// TwinCAT 3 PLC project PMPS_Prototype_Arbiter
// ProgramVersion: 3.1.4022.1
// libraries:
//   LCLS General, * (SLAC)
//   Tc2_MC2, * (Beckhoff Automation GmbH)
//   Tc2_Standard, * (Beckhoff Automation GmbH)
//   Tc2_System, * (Beckhoff Automation GmbH)
//   Tc2_Utilities, * (Beckhoff Automation GmbH)
//   Tc3_Module, * (Beckhoff Automation GmbH)
//   VisuDialogs, * (System)
//   VisuSymbols,3.5.10.0,System
// project tree:
//   DUTs/ E_ExampleDeviceStates.TcDUT (not stored), ST_BeamParams.TcDUT, ST_BinarySolidAttenuator.TcDUT (not stored), ST_Device.TcDUT, ST_DeviceState.TcDUT, ST_SolidAttenuatorBlade.TcDUT
//   / GlobalTextList.TcGTLO, ImagePool.TcIPO (not stored), PlcTask.TcTTO (not stored), Visualization Manager.TcVMO (not stored)
//   GVLs/ GVL.TcGVL, PMPS_GVL_BeamParams.TcGVL
//   POUs/DeviceImplementationEx1/ FB_ExampleDevice.TcPOU (not stored), FB_ExampleDeviceSM.TcPOU (not stored)
//   POUs/DeviceImplementationEx2/ FB_ExampleDeviceSM_All.TcPOU
//   POUs/HelperFunctions/ F_DifferentBeamParams.TcPOU (not stored), F_SafeBPCompare.TcPOU (not stored), F_SetBeamParams.TcPOU (not stored), F_SetStateParams.TcPOU (not stored)
//   POUs/ MAIN.TcPOU, PMPS_Arbiter.TcPOU
//   POUs/MajorComponents/ FB_BeamClassOutputs.TcPOU, FB_LinearGovernor.TcPOU, BeamParameterTransitionManager.TcPOU (not stored), FB_Arbiter.TcPOU, FB_BeamParamAssertionPool.TcPOU (not stored), FB_LinearDeviceStateTable.TcPOU (not stored)
//   POUs/TestComponents/ FB_AttenuatorSimulator.TcPOU, FB_MachineSimulator.TcPOU (not stored), FB_SolidAttenuator.TcPOU
//   VISUs/ ImagerGUI.TcVIS, Visualization.TcVIS
// real-time tasks:
//   TASK PlcTask: cycle T#1ms, priority 20, ADS port 350
// motion (NC):
//   TASK NC-Task 1 SAF: cycle T#2ms, priority 4, ADS port 501
//   TASK NC-Task 1 SVB: cycle T#10ms, priority 8, ADS port 511
//   AXIS Dev1 (id 1)
//   AXIS Dev 2 (id 2)
// variable links:
//   PMPS_Prototype_Arbiter/PMPS_Prototype_Arbiter Instance <-> NC-Task 1 SAF/Axes/Dev 2
//     PlcTask Inputs/MAIN.fbDev2.stDevice.stAxis.NcToPlc <-> Outputs/ToPlc
//     PlcTask Outputs/MAIN.fbDev2.stDevice.stAxis.PlcToNc <-> Inputs/FromPlc
//   PMPS_Prototype_Arbiter/PMPS_Prototype_Arbiter Instance <-> NC-Task 1 SAF/Axes/Dev1
//     PlcTask Inputs/MAIN.fbDev1.stDevice.stAxis.NcToPlc <-> Outputs/ToPlc
//     PlcTask Outputs/MAIN.fbDev1.stDevice.stAxis.PlcToNc <-> Inputs/FromPlc

// ---- DUTs/ST_BeamParams.TcDUT
TYPE ST_BeamParams :
STRUCT
	// Beam parameters
	// These must be filled in by the caller.
	
	//Note: fAtt is a local parameter, meaning it is distributed to the nearest
	// upstream attenuator component.
	fAtt : REAL := 100; //Requested attenuation %
	
	
	
	//Machine parameters
	nBeamClass	:	BYTE := 16#F;
	nRate	:	UDINT	:= 10; //Pulse-rate
	fPP_mJ : REAL := 20; //Per pulse max energy (mJ)
	fUpper_eV	:	REAL	:= 20000; //Requested max eV
	fLower_eV	:	REAL	:= 0; //Requested lower eV
	reV	:	REAL	:=0; //Photon energy (calculated by undulator gap)
END_STRUCT
END_TYPE

// ---- DUTs/ST_Device.TcDUT
TYPE ST_Device :
STRUCT
	//IO
	stAxis	:	AXIS_REF;
	//The following limit switches must be TRUE or high (ie. NC) to enable that direction of motion
	//The EPICS display should show an inverted indicator to communicate end of travel reached
	i_xLoLim	AT %I*	:	BOOL; //Wire normally-closed
	i_xHiLim	AT %I*	:	BOOL; //Wire normally-closed
	
	//Acuator Parameters
	lrUpperPositionLimit	:	LREAL := 10000000000; //Use in conjuntion with limit switches or set to a huge number to ignore
	lrLowerPositionLimit	:	LREAL := -10000000000; //Use in conjuntion with limit switches or set to a huge number to ignore
	
	xEnable	:	BOOL := TRUE;
	
	//Supervisory System
	
	//MPS Override
	xOverrideMPSLimits	: BOOL := FALSE; //Set true to move beyond MPS limits. Note this will trip beam off.
	
	//Device States
	StateTable		:	FB_LinearDeviceStateTable;
	//astStates	:	ARRAY[0..PMPS_GVL_BeamParams.cnMaxStateArrayLen] OF	ST_DeviceState;
	
	stTransitionState	:	ST_DeviceState; //The transition state might have non-zero beam parameters
	nSafeState			:	UDINT; //State where the device is considered safe
	nTransitionState	:	UDINT;
	
	nRequestedState	:	UDINT; //EPICS control, cleaned (checked against array limits) and deposited in nTargetState
	nTargetState	:	UDINT; //The requested state should be deposited here after cleaning
	nActiveState	:	UDINT; //The last successfully reached state
	
	
END_STRUCT
END_TYPE

// ---- DUTs/ST_DeviceState.TcDUT
TYPE ST_DeviceState :
STRUCT
	
	//Database key
	
	//Parent Device
	sParentDevice	:	STRING;
	
	//State name
	sStateName	:	STRING;
	nStateRef	:	UDINT; //Primary key of device state database
	
	//////////////////
	// This stuff may belong in a sub-class or something
	//Position
	rPosition	:	REAL := 0;
	//Tolerance
	rTolerance :	REAL := 0; //+/- amount
	//////////////////
	//Required beam parameters
	stReqBeamParam	:	ST_BeamParams;

END_STRUCT
END_TYPE

// ---- DUTs/ST_SolidAttenuatorBlade.TcDUT
TYPE ST_SolidAttenuatorBlade :
STRUCT
	xRequestedIn	:	BOOL;
	xCurrentIn	:	BOOL;
	rThickness	:	REAL;
END_STRUCT
END_TYPE

// ---- GVLs/GVL.TcGVL

VAR_GLOBAL
	fbArbiter	:	FB_Arbiter;
	g_rTestingVelocity	:	LREAL := VISIBLE_TEST_VELOCITY;
END_VAR

VAR_GLOBAL CONSTANT
	EXCLUDED_ASSERTION_ID	:	UDINT	:= 16#FFFFFFFF; //An assertion ID that should always return "not found" in the assertion pool
	VISIBLE_TEST_VELOCITY	:	LREAL	:= 10;
	FAST_TEST_VELOCITY		:	LREAL	:= 100;
	MAX_DEVICE_STATES		:	UDINT	:= 300;
END_VAR

// ---- GVLs/PMPS_GVL_BeamParams.TcGVL
{attribute 'qualified_only'}
VAR_GLOBAL
	stReqFBDBeamParamsSum	:	ST_BeamParams;
	stReqMethBeamParamSum	:	ST_BeamParams;
	stCurrentBeamParameters	:	ST_BeamParams;
END_VAR
VAR_GLOBAL CONSTANT
	cstFullBeam	:	ST_BeamParams := (
		fAtt := 0,
		fPP_mJ := 1E4,
		fUpper_eV := 1E4,
		fLower_eV := 0,
		nRate	:= UDINT#1000000,
		
);
	cstSafeBeam	:	ST_BeamParams := (
		fAtt := 100,
		fPP_mJ := 0,
		fUpper_eV := 0,
		fLower_eV := 0,
		nRate	:= 0
);
	cnMaxStateArrayLen : INT := 20;
	
	MAX_ASSERIONS	:	UDINT := 100; //Maximum number of assertions permitted in the arbiter
END_VAR

// ---- POUs/MajorComponents/FB_Arbiter.TcPOU
(* FB Arbiter

The arbiter primary objectives are:
- Provide a simple interface for devices to request beam parameter sets
- Provide a way for devices to verify their BPS is active in the arbiter
- Provide a way for devices remove their requests from evaluation
- Evaluate all active beam parameter requests registered with the aribiter,
to determine the safest combination of all sets, provide this set as an output.
- Do all of this with minimal overhead

To these ends, the arbiter uses a hash-table, the rows being a state-id as the key, and a corresponding
 beam parameter set to be evaluated against all the other sets (or rows), in the table.
 
The hash table can be thought of as an array on steriods, they are worth reading about, suffice to say
the hash table will tell you when you reach the end of all the entries, and enables us to find entries quickly.

These features efficiently address the addition, removal, and verification of beam parameter sets listed in the above requirements.

An important thing to pay attention to is the A_Arbitrate action. This action implements the evaluation of beam parameter
sets against each other.

*)

FUNCTION_BLOCK FB_Arbiter
VAR_INPUT
	i_nStateID	:	UDINT; //Set to the stateID of the state requesting the beam parameter set
	i_stAssertBeamParams	:	ST_BeamParams; //Set to the beam parameter set of the state required
END_VAR
VAR_OUTPUT
	q_stBeamParams	:	ST_BeamParams; //Updated on each cycle of the arbiter FB with the current arbitrated beam parameter set
	
	q_xStateIDFound	:	BOOL; //Set true if a state-id is found in the assertion pool after calling A_VerifyAssertion
END_VAR
VAR
	
	fbBPAssertionPool	:	FB_BeamParamAssertionPool; //Table of active beam parameter assertions
	
	getPosPtr	: POINTER TO T_HashTableEntry := 0; 
	getBPStruct	:	ST_BeamParams;
	stOutputBP	:	ST_BeamParams; //Safest beam parameters from all in the assertion pool
	
	
END_VAR

//Arbitrate
(*
This step cycles through every hash table entry, comparing
the beam parameters from each assertion to what we're planning
to assert.

The safer of the two parameters is kept so at the end we may
have a mix of beam parameters, the composition being safe for
all asserters.

*)

//Safest parameters to start
stOutputBP := F_SetBeamParams(
	fAtt := 100,
	fPP_mJ := 0,
	fLower_eV := 0,
	fUpper_eV := 1800,
	nRate := 0
	);

fbBPAssertionPool.A_GetFirst( putPosPtr := 0, getPosPtr=>getPosPtr, getValue=>getBPStruct );
IF fbBPAssertionPool.bOk THEN
	
	//The first entry in the hash table is taken as the setting to arbitrate against
	stOutputBP := F_SetBeamParams(
		fAtt := getBPStruct.fAtt,
		fPP_mJ := getBPStruct.fPP_mJ,
		fLower_eV := getBPStruct.fLower_eV,
		fUpper_eV := getBPStruct.fUpper_eV,
		nRate := getBPStruct.nRate
	);

	REPEAT
		fbBPAssertionPool.A_GetNext( putPosPtr := fbBPAssertionPool.getPosPtr , getPosPtr=>getPosPtr, getValue=>getBPStruct );
		IF fbBPAssertionPool.bOk THEN
			A_Arbitrate();
		END_IF
	UNTIL NOT fbBPAssertionPool.bOk
	END_REPEAT

END_IF

q_stBeamParams := stOutputBP;

ACTION A_Arbitrate:

//Attenuation
//Add something here to register the key that won for each param
stOutputBP.fAtt := MAX(stOutputBP.fAtt, getBPStruct.fAtt);

//Pulse energy
stOutputBP.fPP_mJ := MIN(stOutputBP.fPP_mJ, getBPStruct.fPP_mJ);

//Photon energy ranges
stOutputBP.neVReqRange := stOutputBP.neVReqRange AND getBPStruct.neVReqRange;

//Rate
stOutputBP.nRate := MIN(stOutputBP.nRate, getBPStruct.nRate);
END_ACTION

ACTION A_AssertBP:
//fbTable.A_Add( key := 12345, putValue := putValue, getPosPtr=>getPosPtr, getValue=>getValue );

(* This action adds a state-id and beam parameter set to the beam parameter assertion pool (arbiter
hash table). Use like so:

fbArbiter.A_AssertBP(
i_nStateID := nStateID,
i_stAssertBeamParams := stDesiredBeamParams
);

*)

IF i_nStateID <> EXCLUDED_ASSERTION_ID THEN

	fbBPAssertionPool.A_Add(
		key := i_nStateID,
		putValue := i_stAssertBeamParams,
		getPosPtr=>getPosPtr,
		getValue => getBPStruct
	);
END_IF
	
IF NOT fbBPAssertionPool.bOk THEN
	; //Overflow <TODO>
END_IF
END_ACTION

ACTION A_Init:
// Clears the entire beam parameter assertion pool (hashtable).

fbBPAssertionPool.A_Reset();
END_ACTION

ACTION A_RemoveAssertion:

(* Searches for a state-id, and removes it from the assertion pool.

Use like so:
fbArbiter.A_RemoveAssertion(
i_nStateId := nStateIDAssertionToRemove
);

*)

IF i_nStateId <> EXCLUDED_ASSERTION_ID THEN
	fbBPAssertionPool.A_Remove(key := i_nStateId, getPosPtr=>getPosPtr, getValue=>getBPStruct);
	
	IF fbBPAssertionPool.bOk THEN
		;
	ELSE
		;
	END_IF
END_IF
END_ACTION

ACTION A_VerifyAssertion:

(* Searches state assertion pool for a state-id, and sets q_xStateIDFound true if found.

Use like so:

fbArbiter.A_VerifyAssertion(
i_nStateId := nStateIDAssertionToCheck
);

IF fbArbiter.q_xStateIDFound THEN:
	Do something
ELSE:
	Don't do something

*)

IF i_nStateID <> EXCLUDED_ASSERTION_ID THEN
	
	fbBPAssertionPool.A_Lookup( key := i_nStateID, getPosPtr=>getPosPtr, getValue=>getBPStruct );

	q_xStateIDFound	:= fbBPAssertionPool.bOk;

ELSE
	q_xStateIDFound := FALSE;
END_IF
END_ACTION

END_FUNCTION_BLOCK

// ---- POUs/DeviceImplementationEx2/FB_ExampleDeviceSM_All.TcPOU
(* This version of the block is self contained. Minimizes wiring.*)
FUNCTION_BLOCK FB_ExampleDeviceSM_All
VAR_INPUT
	cBase: UDINT;
END_VAR
VAR_OUTPUT
END_VAR
VAR_IN_OUT
	
END_VAR
VAR
	stDevice	:	ST_Device;
	fbGovernor	:	FB_LinearGovernor;
	mcPower	:	MC_Power;
	mcStop: MC_Stop;
	mcAbsolute	:	MC_MoveAbsolute;
	fbBPTM	:	BeamParameterTransitionManager;
	xStartMove: BOOL;
	
	stCheckState: ST_DeviceState;
	stTargetState	:	ST_DeviceState; //Target device state

END_VAR
VAR PERSISTENT
	nLastActiveState	:	UDINT;
END_VAR

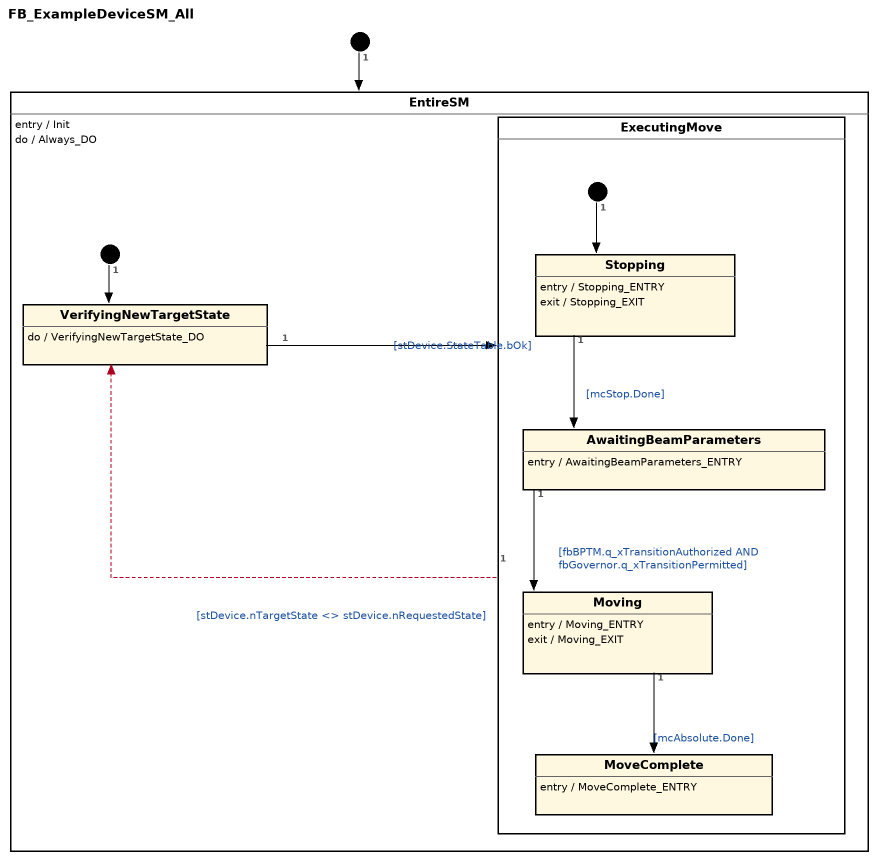
STATECHART FB_ExampleDeviceSM_All  // abortable
    START StartState3
    COMPOSITE STATE EntireSM
        entry / Init
        do / Always_DO
        START StartState1
        COMPOSITE STATE ExecutingMove
            START StartState2
            STATE Stopping
                entry / Stopping_ENTRY
                exit / Stopping_EXIT
            STATE AwaitingBeamParameters
                entry / AwaitingBeamParameters_ENTRY
            STATE Moving
                entry / Moving_ENTRY
                exit / Moving_EXIT
            STATE MoveComplete
                entry / MoveComplete_ENTRY
            StartState2 -> Stopping  // priority 1, on completion
            Stopping -> AwaitingBeamParameters [mcStop.Done] // priority 1, rising edge
            AwaitingBeamParameters -> Moving [fbBPTM.q_xTransitionAuthorized AND fbGovernor.q_xTransitionPermitted] // priority 1, rising edge
            Moving -> MoveComplete [mcAbsolute.Done] // priority 1, rising edge
        END_STATE
        STATE VerifyingNewTargetState
            do / VerifyingNewTargetState_DO
        StartState1 -> VerifyingNewTargetState  // priority 1, on completion
        ExecutingMove -> VerifyingNewTargetState [stDevice.nTargetState <> stDevice.nRequestedState] // priority 1, exception, rising edge
        VerifyingNewTargetState -> ExecutingMove [stDevice.StateTable.bOk] // priority 1
    END_STATE
    StartState3 -> EntireSM  // priority 1, on completion
END_STATECHART

ACTION Always_DO:
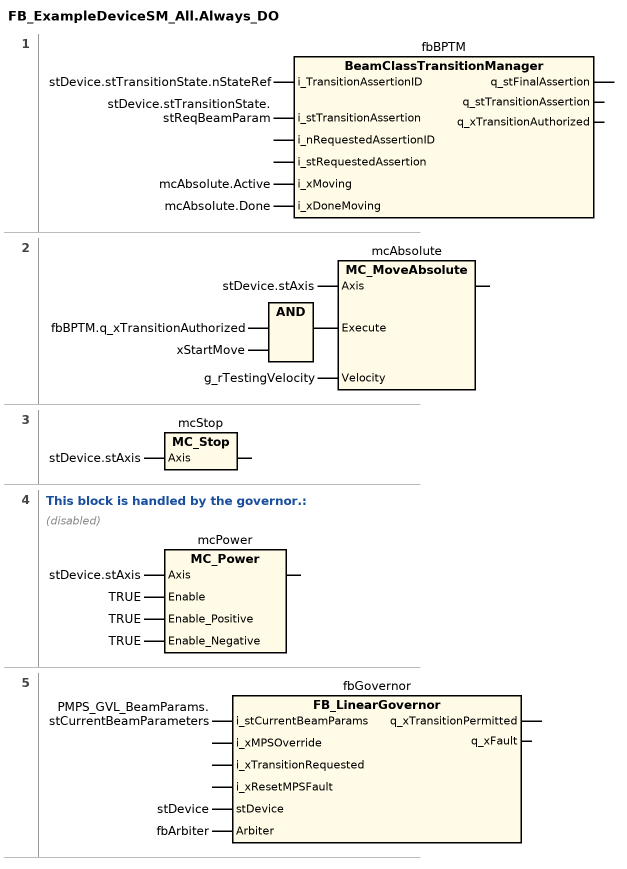
// NETWORK 1
fbBPTM(
    i_TransitionAssertionID := stDevice.stTransitionState.nStateRef,
    i_stTransitionAssertion := stDevice.stTransitionState.stReqBeamParam,
    i_xMoving := mcAbsolute.Active,
    i_xDoneMoving := mcAbsolute.Done); // BeamClassTransitionManager

// NETWORK 2
mcAbsolute(
    Axis := stDevice.stAxis,
    Execute := fbBPTM.q_xTransitionAuthorized AND xStartMove,
    Velocity := g_rTestingVelocity); // MC_MoveAbsolute

// NETWORK 3
mcStop(Axis := stDevice.stAxis); // MC_Stop

// NETWORK 4 (disabled)
// label: This block is handled by the governor.
// mcPower(Axis := stDevice.stAxis, Enable := TRUE, Enable_Positive := TRUE, Enable_Negative := TRUE); // MC_Power

// NETWORK 5
fbGovernor(
    i_stCurrentBeamParams := PMPS_GVL_BeamParams.stCurrentBeamParameters,
    stDevice := stDevice,
    Arbiter := fbArbiter); // FB_LinearGovernor
END_ACTION

ACTION AwaitingBeamParameters_ENTRY:
fbBPTM.i_stRequestedAssertion := stTargetState.stReqBeamParam;
fbBPTM.i_nRequestedAssertionID := stTargetState.nStateRef;

//Tell the governor that we're trying to move.
fbGovernor.i_xTransitionRequested := TRUE;
END_ACTION

ACTION Init:

//Safe State
stDevice.nSafeState := cBase;
stDevice.nTransitionState := cBase+100;

//Initialize the State Table
stDevice.StateTable.A_Reset();

//Device State Table Instantiation
F_SetStateParams(
	nStateRef := stDevice.nSafeState,
	rPosition := 0,
	rTolerance := 10,
	stBeamParams := PMPS_GVL_BeamParams.cstFullBeam,
	Table := stDevice.StateTable
);
F_SetStateParams(
	nStateRef := cBase + 1,
	rPosition := 100,
	rTolerance := 10,
	stBeamParams := F_SetBeamParams(
		fAtt := 20,
		fPP_mJ := 1,
		fLower_eV := 0,
		fUpper_eV := 1500,
		nRate := 10
		),
	Table := stDevice.StateTable
);
F_SetStateParams(
	nStateRef := cBase + 2,
	rPosition := 200,
	rTolerance := 10,
	stBeamParams := F_SetBeamParams(
		fAtt := 30,
		fPP_mJ := 1,
		fLower_eV := 0,
		fUpper_eV := 1500,
		nRate := 10
		),
	Table := stDevice.StateTable
);
F_SetStateParams(
	nStateRef := cBase + 3,
	rPosition := 300,
	rTolerance := 10,
	stBeamParams := F_SetBeamParams(
		fAtt := 20,
		fPP_mJ := 1,
		fLower_eV := 0,
		fUpper_eV := 1500,
		nRate := 10
		),
	Table := stDevice.StateTable
);

F_SetStateParams(
	nStateRef := stDevice.nTransitionState,
	rPosition := 300,
	rTolerance := 10,
	stBeamParams := F_SetBeamParams(
		fAtt := 100,
		fPP_mJ := 0,
		fLower_eV := 0,
		fUpper_eV := 1500,
		nRate := 0
		),
	Table := stDevice.StateTable
);

stDevice.StateTable.A_Lookup(
	key := stDevice.nTransitionState,
	getValue => stDevice.stTransitionState
);

//Need an initialization routine for setting the active state
//Check if the device is at the last known state
//If the device is within the state boundaries, it's considered to be in that state
stDevice.StateTable.A_Lookup(key:= nLastActiveState);
IF stDevice.StateTable.bOk THEN
	stCheckState := stDevice.StateTable.getValue;
ELSE
	stCheckState := stDevice.stTransitionState; //This needs to be safer <TODO>
END_IF

IF stDevice.stAxis.NcToPlc.ActPos <= stCheckstate.rPosition + stCheckState.rTolerance AND
	stDevice.stAxis.NcToPlc.ActPos >= stCheckState.rPosition - stCheckState.rTolerance THEN
	stDevice.nActiveState := nLastActiveState;
ELSE
	stDevice.nActiveState := stDevice.nTransitionState;
END_IF

//Simulation Hardware Limit Switches
stDevice.i_xHiLim := TRUE;
stDevice.i_xLoLim := TRUE;
END_ACTION

ACTION Initialize:

END_ACTION

ACTION MoveComplete_ENTRY:
//Clear transition request
fbGovernor.i_xTransitionRequested := FALSE;
//Latch active state
stDevice.nActiveState := stDevice.nTargetState;
nLastActiveState := stDevice.nActiveState;
END_ACTION

ACTION Moving_ENTRY:
xStartMove := TRUE;
mcAbsolute.Position := stTargetState.rPosition;
END_ACTION

ACTION Moving_EXIT:
xStartMove := FALSE;
END_ACTION

ACTION NewMove_ENTRY:

END_ACTION

ACTION Stopping_ENTRY:
mcStop.Execute := TRUE;
END_ACTION

ACTION Stopping_EXIT:
mcStop.Execute := FALSE;
END_ACTION

ACTION VerifyingNewTargetState_DO:
stDevice.StateTable.A_Lookup(
	key := stDevice.nRequestedState
);

IF stDevice.StateTable.bOk THEN
	stTargetState := stDevice.StateTable.getValue;
	stDevice.nTargetState := stDevice.nRequestedState;
ELSE
	; //log ignored state/ generate an error? <TODO>
END_IF
END_ACTION

END_FUNCTION_BLOCK

// ---- POUs/MajorComponents/FB_LinearGovernor.TcPOU

(* The governor is meant to check your work and keep you from making mistakes.

Checks:
Does your state match the device position and visa versa?
Are the beam parameters safe for the device state?
Did you properly assert the transition and final beam parameters?

*)
FUNCTION_BLOCK FB_LinearGovernor
VAR_INPUT
	i_stCurrentBeamParams	:	ST_BeamParams; //Link to global beam params
	i_xMPSOverride			:	BOOL; //True releases MPS limits after a delay
	i_xTransitionRequested	:	BOOL; //Set true to request a transition
	i_xResetMPSFault	:	BOOL; //Set true to clear MPS fault 
END_VAR
VAR_OUTPUT
	q_xTransitionPermitted	:	BOOL; //True when governor has released restrictions
	q_xFault	:	BOOL; //Set if MC_Power has an error, or override mode is requested
END_VAR
VAR_IN_OUT
	stDevice	:	ST_Device; //The governed
	Arbiter	:	FB_Arbiter;
END_VAR
VAR
	mcPower	:	MC_Power;
	
	xActuatorPositiveEnable: BOOL;
	xActuatorNegativeEnable: BOOL;
	
	xMPSPositiveEnable	:	BOOL;
	xMPSNegativeEnable	:	BOOL;
	lrPosition: LREAL;
	
	lrLatchedTargetPosition	:	LREAL;
	lrLatchedTargetTolerance	:	LREAL;
	
	lrMPSUpperLimit: LREAL;
	lrMPSLowerLimit: LREAL;
	rtNewState: R_TRIG;
	xTransitionOK: BOOL;
	
	tonMPSOverrideMode	:	TON := (
		PT := T#5S
	);
	
	srMPSFault	:	SR;
	// Actuator out of bounds fault
	xActuatorOOB: BOOL;
	//Beam parameters out of spec
	xBeamParamsOOS: BOOL;
	//Beam parameters of currently latched state
	
	stLatchedBeamParams: ST_BeamParams;
	stTargetState: ST_DeviceState;
	
	rtLatchNewState	:	R_TRIG;
	xInit: BOOL := TRUE;
	
	stInitDeviceState: ST_DeviceState;
	// Indicates an error with initialization
	xInitFault: BOOL;
	// Indicates the state could not be found in the state table. There may be something wrong in the device state machine implementation or state table instantiation.
	xStateLookupError: BOOL;
END_VAR


lrPosition := stDevice.stAxis.NcToPlc.ActPos; //Actuator position

stDevice.stAxis.ReadStatus();
//Init
////////////////////////////////
	IF xInit THEN
		xInit := FALSE;
		stDevice.StateTable.A_Lookup(key := stDevice.nActiveState);
		IF stDevice.StateTable.bOk THEN
			stInitDeviceState := stDevice.StateTable.getValue;
			xInitFault := FALSE;
		ELSE
			xInitFault := TRUE;
		END_IF
		lrLatchedTargetPosition := stInitDeviceState.rPosition;
		lrLatchedTargetTolerance := stInitDeviceState.rTolerance;
		stLatchedBeamParams := stInitDeviceState.stReqBeamParam;
	END_IF

// The governor will permit transitions once it verifies the transition assertion is active
// Note the governor does not verify the target state beam params are asserted, perhaps it should <TODO>
////////////////////////////////
	IF i_xTransitionRequested THEN
		Arbiter.A_VerifyAssertion(
			i_nStateID := stDevice.stTransitionState.nStateRef
		);
		xTransitionOK := Arbiter.q_xStateIDFound AND F_SafeBPCompare(PMPS_GVL_BeamParams.stCurrentBeamParameters, stDevice.stTransitionState.stReqBeamParam);
		
		//Set the target state for evaluation in further logic
		stdevice.StateTable.A_Lookup(key := stDevice.nTargetState);
		IF stDevice.StateTable.bOk THEN
			stTargetState := stDevice.StateTable.getValue;
			xStateLookupError := FALSE;
		ELSE
			xStateLookupError := TRUE;
		END_IF
	ELSE
		xTransitionOK := FALSE;
	END_IF

(* Note about TransitionRequested

If TransitionRequested goes false during a transition, an MPS fault may be induced. This occurs
because the Actuator Out of Bounds fault will go back to using the original state limits, which
the axis may have already moved beyond.

To avoid this transient fault, make sure your device state machine is implemented such that the 
transition request to the governor block remains high until the target position is reached.
*)

//Determine if a transition is complete and latch the new state
(* A transition is complete when:

Axis at standstill.
Axis within tolerance.
No transition req.

Once these conditions are met, the MPS limits shall re-engage to restrict the
axis motion to the tolerance around the state position and the MPS fault monitors
shall evaluate based on the newly latched target state.
*)

rtLatchNewState(CLK := stDevice.stAxis.Status.StandStill AND
	lrPosition <= stTargetState.rPosition + stTargetState.rTolerance AND
	lrPosition >= stTargetState.rPosition - stTargetState.rTolerance AND
	NOT i_xTransitionRequested);
	
IF rtLatchNewState.Q THEN
	lrLatchedTargetPosition := stTargetState.rPosition;
	lrLatchedTargetTolerance := stTargetState.rTolerance;
	stLatchedBeamParams := stTargetState.stReqBeamParam;
END_IF

//Let other blocks know the governor won't interfer with transitions
q_xTransitionPermitted := xTransitionOK;

//Adjust limit ranges based on active state and current target
IF xTransitionOK THEN
	//Extend range to include target state
	lrMPSUpperLimit := MAX(lrMPSUpperLimit, stTargetState.rPosition + stTargetState.rTolerance);
	lrMPSLowerLimit := MIN(lrMPSLowerLimit, stTargetState.rPosition - stTargetState.rTolerance);
ELSE
	//Calculate the limit positions for MPS based on current state
	lrMPSUpperLimit := lrLatchedTargetPosition + lrLatchedTargetTolerance;
	lrMPSLowerLimit := lrLatchedTargetPosition - lrLatchedTargetTolerance;
END_IF

//MPS Faults
//Fault if the beam is unsafe for current state
xBeamParamsOOS := NOT F_SafeBPCompare(PMPS_GVL_BeamParams.stCurrentBeamParameters, stLatchedBeamParams);

//Fault if the position is outside of the permitted range
xActuatorOOB := lrPosition >= lrMPSUpperLimit OR lrPosition <= lrMPSLowerLimit;



//Latch the MPS faults
srMPSFault.SET1 := xActuatorOOB OR xBeamParamsOOS OR xStateLookupError;
srMPSFault(RESET:=i_xResetMPSFault); 

(* Note: The state lookup error is recoverable, because a different target state might be valid.
*)


//MPS override
(* In override mode, the device will be free to move anywhere within it's travel range *)
//Permit motion after a small delay
tonMPSOverrideMode(IN:=i_xMPSOverride OR stDevice.xOverrideMPSLimits);

//Virtual limit switch evaluation
xActuatorPositiveEnable	:= stDevice.i_xHiLim AND lrPosition <= stDevice.lrUpperPositionLimit;
xActuatorNegativeEnable	:= stDevice.i_xLoLim AND lrPosition >= stDevice.lrLowerPositionLimit;

//Evaluate MPS limit states
xMPSPositiveEnable := lrPosition <= lrMPSUpperLimit;
xMPSNegativeEnable := lrPosition >= lrMPSLowerLimit;

//Final Limit switch evaluation
mcPower.Enable_Positive := xActuatorPositiveEnable AND (tonMPSOverrideMode.Q OR xMPSPositiveEnable);
mcPower.Enable_Negative := xActuatorNegativeEnable AND (tonMPSOverrideMode.Q OR xMPSNegativeEnable);

mcPower(
	Axis := stDevice.stAxis,
	Enable := stDevice.xEnable //link to device enable <TODO>
);

//An mcPower error or MPS override, or MPS fault, produces a fault.
q_xFault := mcPower.Error OR i_xMPSOverride OR srMPSFault.Q1 OR xInitFault;

END_FUNCTION_BLOCK

// ---- POUs/MAIN.TcPOU
PROGRAM MAIN
VAR
	fbDev1	:	FB_ExampleDeviceSM_All;
	fbDev2	:	FB_ExampleDeviceSM_All;
	
	BP1	:	ST_BeamParams;
	BP2	:	ST_BeamParams;
	Test	:	BOOL;
	
	rtInit	:	R_TRIG;
	Initialize	:	BOOL := TRUE;
	
	
	FB_ExampleDeviceSM_All_0: FB_ExampleDeviceSM_All;
	FB_ExampleDeviceSM_All_1: FB_ExampleDeviceSM_All;
END_VAR

//Sub-system Device PLC
// This PLC runs 4 

Test := F_SafeBPCompare(BP1,BP2);

IF Initialize THEN
	fbDev1(cBase := 10);
	fbDev2(cBase := 1000);
	fbArbiter.A_Init();
	Initialize := FALSE;
END_IF

//Example devices
fbDev1();
fbDev2();

PMPS_Arbiter();

ACTION FB_Vis:
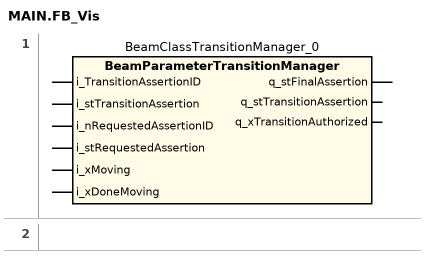
// NETWORK 1
BeamClassTransitionManager_0(); // BeamParameterTransitionManager

// NETWORK 2
END_ACTION

ACTION Initialize:

END_ACTION

END_PROGRAM

// ---- POUs/PMPS_Arbiter.TcPOU
PROGRAM PMPS_Arbiter
VAR
	
	
	fbMachine	:	FB_MachineSimulator;
END_VAR


//Execute arbiter
fbArbiter();

//Machine simulator
fbMachine(
	i_stAssertedParams := fbArbiter.q_stBeamParams,
	q_stMachineParams => PMPS_GVL_BeamParams.stCurrentBeamParameters
	);

END_PROGRAM

// ---- POUs/MajorComponents/FB_BeamClassOutputs.TcPOU
(*
Sets the beam class assertion lines for a given beam class.
*)
FUNCTION_BLOCK FB_BeamClassOutputs
VAR_INPUT
	i_ArbiterBP	:	ST_BeamParams;
END_VAR
VAR_OUTPUT
END_VAR
VAR
	wBeamClass	:	BYTE;
	q_BC_ASSERTION_LINES	AT	%Q*	: ARRAY [1..16] OF	BOOL;
	InitCounter: INT;
	counter	:	INT;
END_VAR


//Beam Class
////////////////////////////////////
//0x0 = 0000 0000 0000 0000
//0x1 = 0000 0000 0000 0001
//0xF = 1111 1111 1111 1111

//Initialize BC lines to zero on every pass
FOR InitCounter := 1 TO 16 DO
	q_BC_ASSERTION_LINES[InitCounter] := FALSE;
END_FOR

//Set BC lines according to beam class
//A BC of 0x0 would pass over this loop, setting none of the lines high
// , as FOR loops check the initialized variable at the top to see if it's >
// than the "TO" variable.
FOR wBeamClass:=1 TO i_ArbiterBP.nBeamClass DO
	q_BC_ASSERTION_LINES[wBeamClass] := TRUE;
END_FOR

END_FUNCTION_BLOCK

// ---- POUs/TestComponents/FB_AttenuatorSimulator.TcPOU
FUNCTION_BLOCK FB_AttenuatorSimulator
VAR_INPUT
	i_rRequestedAttenuation	:	REAL;
END_VAR
VAR_OUTPUT
	q_xFault	:	BOOL;
	q_rCurrentAttenuation	:	REAL;
END_VAR
VAR_IN_OUT
	Arbiter	:	FB_Arbiter; //Higher level arbiter from which upstream attenuation can be requested
END_VAR
VAR
	tonDelay	:	TON := (
		PT := T#3S
		);
	rLower_eVThreshold	:	REAL := 300;
END_VAR

// Really basic delay
tonDelay(IN := i_rRequestedAttenuation <> q_rCurrentAttenuation);

IF tonDelay.Q THEN
	q_rCurrentAttenuation := i_rRequestedAttenuation;
END_IF

END_FUNCTION_BLOCK

// ---- POUs/TestComponents/FB_SolidAttenuator.TcPOU
FUNCTION_BLOCK FB_SolidAttenuator
VAR_INPUT
	i_rRequestedAttenuation	:	REAL;
END_VAR
VAR_OUTPUT
	q_xFault	:	BOOL;
	q_rCurrentAttenuation	:	REAL;
END_VAR
VAR_IN_OUT
	Arbiter	:	FB_Arbiter; //Higher level arbiter from which upstream attenuation can be requested
END_VAR
VAR
	stAttenuator	:	ST_BinarySolidAttenuator;
	nSearchStart: INT;
	nArrayLength: INT;
	axNewBladeStates	:	ARRAY [0..9]	OF	BOOL;
	nTryIndex: INT;
	rCurrentAccumulatedAttenuation: REAL;
	rTryFilter: REAL;
	rTryAttenuation: REAL;
	rRequestedAttenuation: REAL;
END_VAR



//

//Assuming the blades are ordered thickest to thinnest 
REPEAT
	rTryAttenuation := rCurrentAccumulatedAttenuation + stAttenuator.axBlades[nTryIndex].rThickness;
	IF rRequestedAttenuation >= rTryAttenuation THEN
		rCurrentAccumulatedAttenuation := rTryAttenuation;
		axNewBladeStates[nTryIndex] := TRUE;
	ELSE
		axNewBladeStates[nTryIndex] := FALSE;
	END_IF
UNTIL
	nTryIndex >= nArrayLength
END_REPEAT

END_FUNCTION_BLOCK

// ---- GlobalTextList.TcGTLO
TEXTLIST GlobalTextList
  108 = '%3.2f'
  632 = '%d'
  511 = 'Arbiter Assertions'
  482 = 'Arbiter Stats'
  300 = 'Assertion Count'
  843 = 'Assertion ID'
  826 = 'Assertion Pool'
  68 = 'Assertion Pool State'
  766 = 'Assertion Pool Stats'
  708 = 'Att'
  276 = 'Attenuation'
  796 = 'Free Slots'
  100 = 'GroupBox'
  284 = 'Imager'
  447 = 'Imager 1'
  330 = 'Imager 2'
  870 = 'lock'
  217 = 'Lower eV'
  585 = 'Machine Parameters'
  419 = 'MPS Override'
  967 = 'MPS Upper Limit'
  682 = 'NA'
  950 = 'nStateRef'
  934 = 'Photon Energy'
  667 = 'pNext'
  410 = 'PPE'
  650 = 'Pulse Energy'
  479 = 'Rate'
  326 = 'rPosition'
  509 = 'rTolerance'
  140 = 'sParentDevice'
  915 = 'sStateName'
  29 = 'State 1'
  57 = 'State 2'
  955 = 'State 3'
  290 = 'State Control'
  553 = 'stReqBeamParam'
  13 = 'Upper eV'
  396 = 'value'
END_TEXTLIST

// ---- VISUs/ImagerGUI.TcVIS
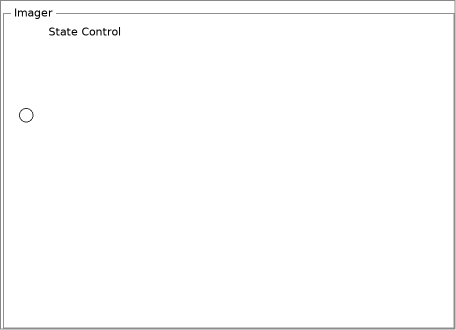
VISUALIZATION ImagerGUI  // 456x330
VAR_IN_OUT
	fbDev	:	FB_ExampleDevice;
END_VAR
    GroupBox (3,5 451x323), "Imager"
        RadioButton (14,49 97x122), variable: fbDev.stDevice.nRequestedState
            Areas[1]: Text=State 1
            Areas[2]: Text=State 2
            Areas[3]: Text=State 3
        Label (7,12 150x30), "State Control"
END_VISUALIZATION

// ---- VISUs/Visualization.TcVIS
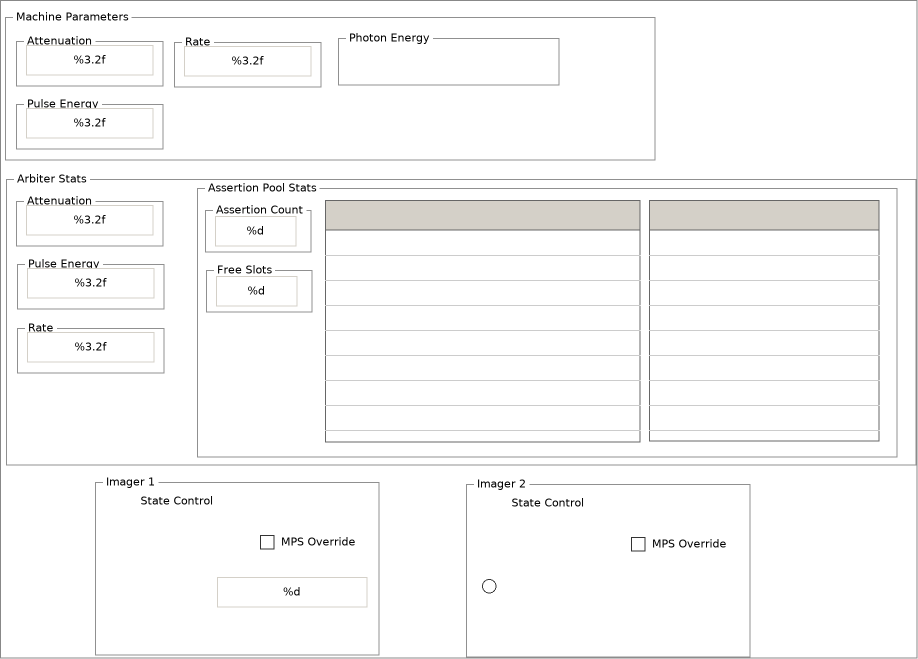
VISUALIZATION Visualization  // 918x659
    GroupBox (5,9 650x151), "Machine Parameters"
        GroupBox (11,24 147x53), "Attenuation"
            Textfield (10,12 127x30), "%3.2f", text variable: PMPS_GVL_BeamParams.stCurrentBeamParameters.fAtt
        GroupBox (11,87 147x53), "Pulse Energy"
            Textfield (10,12 127x30), "%3.2f", text variable: PMPS_GVL_BeamParams.stCurrentBeamParameters.fPP_mJ
        GroupBox (169,25 147x53), "Rate"
            Textfield (10,12 127x30), "%3.2f", text variable: PMPS_GVL_BeamParams.stCurrentBeamParameters.nRate
        GroupBox (333,21 221x55), "Photon Energy"
    GroupBox (6,171 910x294), "Arbiter Stats"
        GroupBox (191,9 700x277), "Assertion Pool Stats"
            GroupBox (9,82 106x50), "Free Slots"
                Textfield (10,14 81x30), "%d", text variable: fbArbiter.fbBPAssertionPool.hTable.nFree
            GroupBox (8,22 106x50), "Assertion Count"
                Textfield (10,14 81x30), "%d", text variable: fbArbiter.fbBPAssertionPool.hTable.nCount
            Table (128,20 315x242), data array: fbArbiter.fbBPAssertionPool.dataPool
                p3854506369: fbArbiter.fbBPAssertionPool.dataPool[INDEX].fAtt
                p1892666644: fbArbiter.fbBPAssertionPool.dataPool[INDEX].fPP_mJ
                p338671338: fbArbiter.fbBPAssertionPool.dataPool[INDEX].fUpper_eV
                p2170511999: fbArbiter.fbBPAssertionPool.dataPool[INDEX].fLower_eV
                p1755163831: Upper eV
                p4092479075: Lower eV
            Table (452,20 230x241), data array: fbArbiter.fbBPAssertionPool.entries
                p3854506369: fbArbiter.fbBPAssertionPool.entries[INDEX].key
                p1892666644: fbArbiter.fbBPAssertionPool.entries[INDEX].value
                p338671338: fbArbiter.fbBPAssertionPool.entries[INDEX].lock
                p2170511999: fbArbiter.fbBPAssertionPool.entries[INDEX].pNext
                p3723444502: fbArbiter.fbBPAssertionPool.entries[INDEX].pNextFree
                p1218418051: fbArbiter.fbBPAssertionPool.entries[INDEX].pNextGlob
                p2232123230: Assertion ID
        GroupBox (10,22 147x53), "Attenuation"
            Textfield (10,12 127x30), "%3.2f", text variable: fbArbiter.q_stBeamParams.fAtt
        GroupBox (11,85 147x53), "Pulse Energy"
            Textfield (10,12 127x30), "%3.2f", text variable: fbArbiter.q_stBeamParams.fPP_mJ
        GroupBox (11,149 147x53), "Rate"
            Textfield (10,12 127x30), "%3.2f", text variable: fbArbiter.stOutputBP.nRate
    GroupBox (466,476 284x181), "Imager 2"
        RadioButton (14,49 97x122), variable: MAIN.fbDev2.stDevice.nRequestedState
            Areas[1]: Text=State 1
            Areas[2]: Text=State 2
            Areas[3]: Text=State 3
        Label (7,12 150x30), "State Control"
        Checkbox (163,53 110x30), "MPS Override", variable: MAIN.fbDev2.stDevice.xOverrideMPSLimits
    GroupBox (95,474 284x181), "Imager 1"
        Label (7,12 150x30), "State Control"
        Checkbox (163,53 111x30), "MPS Override", variable: MAIN.fbDev1.stDevice.xOverrideMPSLimits
        Textfield (122,103 150x30), "%d", text variable: MAIN.fbDev1.stDevice.nRequestedState
            OnMouseClick: write the text variable via Default
END_VISUALIZATION
